TYPE PT1T2_Parameter_Strukt :
STRUCT
	K :			REAL;
	T1 :		REAL;
	T2 :		REAL;
END_STRUCT
END_TYPE

(* stored: Version 1.1.0.1, ProductVersion 3.1.4024.13
   DUT PT1T2_Parameter_Strukt: Id {9e9498a9-7c55-4e5e-961d-9e412d523e8c} *)
